// TIA Portal V18 export
DATA_BLOCK "SS2_A3_32DI_DI_Vars"   // DB11141
{ S7_Optimized_Access := 'FALSE' }
VERSION : 0.1
// stored: AutoNumber false, DBAccessibleFromOPCUA true, IsOnlyStoredInLoadMemory false, IsWriteProtectedInAS false
   VAR
      DI1 : "UDT_DIadv";
      DI2 : "UDT_DIadv";
      DI3 : "UDT_DIadv";
      DI4 : "UDT_DIadv";
      DI5 : "UDT_DIadv";
      DI6 : "UDT_DIadv";
      DI7 : "UDT_DIadv";
      DI8 : "UDT_DIadv";
      DI9 { S7_SetPoint := 'True'} : "UDT_DIadv";
      DI10 { S7_SetPoint := 'True'} : "UDT_DIadv";
      DI11 { S7_SetPoint := 'True'} : "UDT_DIadv";
      DI12 { S7_SetPoint := 'True'} : "UDT_DIadv";
      DI13 { S7_SetPoint := 'True'} : "UDT_DIadv";
      DI14 { S7_SetPoint := 'True'} : "UDT_DIadv";
      DI15 { S7_SetPoint := 'True'} : "UDT_DIadv";
      DI16 { S7_SetPoint := 'True'} : "UDT_DIadv";
      DI17 { S7_SetPoint := 'True'} : "UDT_DIadv";
      DI18 { S7_SetPoint := 'True'} : "UDT_DIadv";
      DI19 { S7_SetPoint := 'True'} : "UDT_DIadv";
      DI20 { S7_SetPoint := 'True'} : "UDT_DIadv";
      DI21 { S7_SetPoint := 'True'} : "UDT_DIadv";
      DI22 { S7_SetPoint := 'True'} : "UDT_DIadv";
      DI23 { S7_SetPoint := 'True'} : "UDT_DIadv";
      DI24 { S7_SetPoint := 'True'} : "UDT_DIadv";
      DI25 { S7_SetPoint := 'True'} : "UDT_DIadv";
      DI26 { S7_SetPoint := 'True'} : "UDT_DIadv";
      DI27 { S7_SetPoint := 'True'} : "UDT_DIadv";
      DI28 { S7_SetPoint := 'True'} : "UDT_DIadv";
      DI29 { S7_SetPoint := 'True'} : "UDT_DIadv";
      DI30 { S7_SetPoint := 'True'} : "UDT_DIadv";
      DI31 { S7_SetPoint := 'True'} : "UDT_DIadv";
      DI32 { S7_SetPoint := 'True'} : "UDT_DIadv";
   END_VAR
BEGIN
   DI3.cFuncSystemID := 2;
   DI3.cFuncVar := 0;
   DI4.cFuncSystemID := 2;
   DI4.cFuncVar := 3;
   DI5.cFuncSystemID := 2;
   DI5.cFuncVar := 2;
   DI6.cFuncSystemID := 2;
   DI7.cFuncSystemID := 2;
   DI7.cFuncVar := 14;
   DI8.cFuncSystemID := 2;
   DI9.cFuncSystemID := 2;
   DI9.cFuncVar := 9;
   DI10.cFuncSystemID := 2;
   DI11.cFuncSystemID := 2;
   DI12.cFuncSystemID := 2;
   DI12.cFuncVar := 8;
   DI13.cFuncSystemID := 2;
   DI14.cFuncSystemID := 2;
   DI15.cFuncSystemID := 2;
   DI16.cFuncSystemID := 2;
   DI17.cFuncSystemID := 10;
   DI17.cFuncVar := 35;
   DI18.cFuncSystemID := 10;
   DI18.cFuncVar := 36;
   DI19.cFuncSystemID := 10;
   DI19.cFuncVar := 37;
   DI20.xInversion := true;
   DI20.cFuncSystemID := 10;
   DI20.cFuncVar := 10;
   DI21.xInversion := true;
   DI21.cFuncSystemID := 10;
   DI21.cFuncVar := 13;
   DI22.cFuncSystemID := 10;
   DI22.cFuncVar := 9;
   DI23.cFuncSystemID := 10;
   DI23.cFuncVar := 12;
   DI24.xInversion := true;
   DI24.cFuncSystemID := 10;
   DI24.cFuncVar := 33;
   DI25.cFuncSystemID := 10;
   DI25.cFuncVar := 32;
   DI26.cFuncSystemID := 10;
   DI26.cFuncVar := 14;
   DI27.cFuncSystemID := 10;
   DI27.cFuncVar := 34;
   DI29.cFuncSystemID := 10;
   DI30.cFuncSystemID := 10;
   DI30.cFuncVar := 46;
   DI31.cFuncSystemID := 10;
   DI31.cFuncVar := 44;
END_DATA_BLOCK
